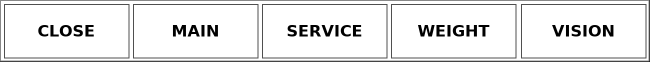
VISUALIZATION vTableWeighingNavigation  // 650x62
VAR_IN_OUT
	fbTableControl: FB_TableControl;
END_VAR
    Rectangle (0,0 650x62)
    Rectangle (391,4 125x54), "WEIGHT"
        OnMouseDown: execute { fbTableControl.stHMI.iDialogNumber:=204; }
    Rectangle (4,4 125x54), "CLOSE"
        OnMouseDown: execute { fbTableControl.stHMI.iDialogNumber:=0; }
    Rectangle (262,4 125x54), "SERVICE"
        OnMouseDown: execute { fbTableControl.stHMI.iDialogNumber:=203; }
    Rectangle (133,4 125x54), "MAIN"
        OnMouseDown: execute { fbTableControl.stHMI.iDialogNumber:=201; }
    Rectangle (521,4 125x54), "VISION"
        OnMouseDown: execute { fbTableControl.stHMI.iDialogNumber:=205; }
END_VISUALIZATION

(* stored: Version 1.1.0.1, ProductVersion 3.1.4024.15
   Visu vTableWeighingNavigation: Id {11cef33d-20c6-40ce-8388-15b5a9e99b9f} *)
